ABB RAPID module: Projet1.mod

MODULE Lab1
! ----------------------------------------------------------------------------
! Programme : GPA546Lab1
! Auteurs : Olivier Millette ET Camilo Serna
! Date : Mai 14, 2024
! Révision : V0.0
!
! Description :
! Ce programme permet de prendre deux blocs dans une glissoire et de les
! superposer sur une table de travail.
! ----------------------------------------------------------------------------

  ! Donnees de type position enseignees
  PERS robtarget rGlissoire:=[[0,0,0],[1,0,0,0],[0,0,0,0],[9E+09,9E+09,9E+09,9E+09,9E+09,9E+09]];
  PERS robtarget rDepot:=[[0,0,0],[1,0,0,0],[0,0,0,0],[9E+09,9E+09,9E+09,9E+09,9E+09,9E+09]];
  PERS robtarget rRetrait:=[[0,0,0],[1,0,0,0],[0,0,0,0],[9E+09,9E+09,9E+09,9E+09,9E+09,9E+09]];

  ! Donnees de type position calculees
  VAR robtarget rDepot2;

  ! Donnees de type constante
  CONST num Epaisseur:= 1; ! Épaisseur d'un bloc (en pouces)
  CONST num PouceToMM:= 25.4; ! Facteur de conversion
  CONST num Decalage:= -80; ! Distance d'approche ou de retrait (mm) Additionnele(ajouter +X pour marge de sécurité)

  ! Données de type Variable
  VAR num EpaisMM:=0;

  ! Vitesse d'approche et de retrait (mm/sec)
  CONST speeddata LowSpeed:=[250,500,5000,1000];

  ! Vitesse maximale du robot (mm/sec)
  CONST speeddata HighSpeed:=[1000,500,5000,1000];

  ! Etat des entrees/sorties
  CONST dionum Ouverte:=0;
  CONST dionum Fermee:=1;
  CONST dionum Retracte:=0;
  CONST dionum Extension:=1;

  ! Variable pour limiter la zone de travail du robot
  VAR wztemporary EspaceRestreint;

! ----------------------------------------------------------------------------
! Procedure : main
! Auteurs : Yanick Noiseux
! Date : 4-08-2011
! Révision : 1.1
! Révision par: Martin Gaudreault
! Description :
! Routine qui est executee par le robot initialement.
! **** elle doit être en mode "cycle"
!
! ----------------------------------------------------------------------------
!**************************************************************************************
PROC main()

	! 1) Initialisation :
	init;

	! Deplacement a la position de repos
	MoveJ rRetrait, HighSpeed, fine, tPince_bloc\wobj:=wobj0;

	! 2) Calculs :
	EpaisMM := Epaisseur * PouceToMM; ! Conversion en mm
	rDepot2 := Offs(rDepot,0,0,-EpaisMM);

	! 3) Déplacement du premier bloc :
	! Prise du bloc dans le glissoire
	Prise;
	! Dépôt du bloc 1 à la localisation rDepot :
	Depot(rDepot);

	! 4) Déplacement du deuxième bloc :
	! Prise du bloc dans le glissoire
	Prise;
	! Dépôt du bloc 2 à la localisation rDepot :
	Depot(rDepot2);

	! 5) Retourner le robot a la position de repos
	MoveJ rRetrait, HighSpeed, fine, tPince_bloc\wobj:=wobj0;

	Pince\Ouvert; ! Ouvrir la pince

ENDPROC
!**************************************************************************************

! ----------------------------------------------------------------------------
! Procedure : init
! Auteurs : Yanick Noiseux
! Date : 4-08-2011
! Révision : 1.1
! Révision par: Martin Gaudreault
! Description :
! Routine qui initialise les variables systèmes et les états des sorties
!
! ----------------------------------------------------------------------------
!**************************************************************************************
PROC init()

	! volume pour limiter les articulation du robot
	VAR shapedata joint_space;

	! Ne garder que les deux constantes correspondant a votre robot
	! Ces valeurs ne doivent pas être changées afin d'aider a la securite et représentent
    ! les limites logicielles pour chacun des axes

	! *** décommentez ces deux lignes si vous êtes sur le robot 1
	!CONST jointtarget low_pos:=[[ 54, -25, -85, -90, -103, -289 ],[ 9E9, 9E9, 9E9, 9E9, 9E9, 9E9 ]];
	!CONST jointtarget high_pos:=[[ 128,  55,  55,  90,  103,  109 ],[ 9E9, 9E9, 9E9, 9E9, 9E9, 9E9 ]];

	! *** décommentez ces deux lignes si vous êtes sur le robot 2
	!CONST jointtarget low_pos:=[[ -134, -25, -85, -90, -103, -289 ],[ 9E9, 9E9, 9E9, 9E9, 9E9, 9E9 ]];
	!CONST jointtarget high_pos:=[[ -65,  55,  55,  90,  103,  109 ],[ 9E9, 9E9, 9E9, 9E9, 9E9, 9E9 ]];

	! *** décommentez ces deux lignes si vous êtes sur le robot 3
	!CONST jointtarget low_pos:=[[ 44, -25, -85, -90, -103, -289 ],[ 9E9, 9E9, 9E9, 9E9, 9E9, 9E9 ]];
	!CONST jointtarget high_pos:=[[ 118,  55,  55,  90,  103,  109 ],[ 9E9, 9E9, 9E9, 9E9, 9E9, 9E9 ]];

	! *** décommentez ces deux lignes si vous êtes sur le robot 4
	!CONST jointtarget low_pos:=[[ -104, -25, -85, -90, -103, -289 ],[ 9E9, 9E9, 9E9, 9E9, 9E9, 9E9 ]];
	!CONST jointtarget high_pos:=[[ -28,  55,  55,  90,  103,  109 ],[ 9E9, 9E9, 9E9, 9E9, 9E9, 9E9 ]];

	! activation de la limitation, obligatoire
	WZFree EspaceRestreint;
	WZLimJointDef \Outside, joint_space, low_pos, high_pos;
	WZLimSup \Temp, EspaceRestreint, joint_space;

	VelSet 25,1000; ! Limitation imposée pour la sécurité, obligatoire

	SetDO DO09_FV0101, Retracte; ! Rentrer le vérin
	Pince\Ouvert; ! Ouvrir la pince

ENDPROC
!**************************************************************************************

! ----------------------------------------------------------------------------
! Procedure : Prise
! Auteurs : Yanick Noiseux
! Date : 4-08-2011
! Révision : 1.0
!
! Description :
! Routine qui s'approche du glissoire, atends une piece,
! l'indexe et la prends de maniere securitaire
!
! ----------------------------------------------------------------------------
!**************************************************************************************
PROC Prise()

! Vérification de présence de bloc dans la glissoire
	IF DI09_ZS0101 = 0 THEN
		TPErase;
		TPWrite "Aucun bloc dans la glissoire";
		TPWrite "Placer deux bloc et remettre en mode AUTO";
		WaitDI DI09_ZS0101, 1; ! Attente d'un bloc
		Waittime 1; ! attente que le bloc se stabilise
	ENDIF

	! Prehension du bloc
	MoveJ RelTool(rGlissoire,0,0,Decalage),HighSpeed,z50,tPince_bloc\wobj:=wobj0;
	SetDO DO09_FV0101, Extension; ! Indexer le bloc durant le mouvement
	WAITDI DI14_ZS0104,1; ! Attendre pour le vérin sortie
	MoveL rGlissoire, LowSpeed, fine, tPince_bloc\wobj:=wobj0;
	Pince\Fermer; ! Fermer la pince
	SetDO DO09_FV0101, Retracte;
	WAITDI DI14_ZS0104,0;
	MoveL RelTool(rGlissoire,0,0,Decalage),LowSpeed,z50,tPince_bloc\wobj:=wobj0;

ENDPROC
!**************************************************************************************

! ----------------------------------------------------------------------------
! Procedure : Depot
! Auteurs : Yanick Noiseux
! Date : 4-08-2011
! Révision : 1.1
! Révision par: Martin Gaudreault
! Description :
! Routine qui initialise les variables systèmes et les états des sorties
!
! Parametre: recoit un robtarget où aller déposer le bloc avec aproche et degagement
!
! ----------------------------------------------------------------------------
!**************************************************************************************
PROC Depot(robtarget rPosDepot) 	! Déclaration de la procédure de dépôt
	! 1) Approche rapide à la position de dépôt, en décalant en Z pour éviter les collisions
	MoveJ RelTool(rPosDepot,0,0,Decalage), HighSpeed, z50, tPince_bloc\wobj:=wobj0;

	! 2) Descente linéaire en mode « fine » à vitesse réduite pour un positionnement précis
	MoveL rPosDepot, LowSpeed, fine, tPince_bloc;

	! 3) Ouverture de la pince pour relâcher le bloc
	Pince\Ouvert; ! Ouvrir la pince

	! 4) Remontée linéaire à la position d’approche (décalée en Z) pour dégager l’outil
	MoveL RelTool(rPosDepot,0,0,Decalage), LowSpeed, z50, tPince_bloc\wobj:=wobj0;

ENDPROC
!**************************************************************************************

! ----------------------------------------------------------------------------
! Procedure : Pince
! Auteurs : Yanick Noiseux
! Date : 4-08-2011
! Révision : 1.1
! Révision par: Martin Gaudreault
! Description :
! Routine qui Défini l'état de l'outil pince du robot
! ----------------------------------------------------------------------------
!**************************************************************************************
PROC Pince(\switch Ouvert | switch Fermer)

    ! Action sur la pince
    IF Present(Fermer) THEN
		! verifie si la sortie doit-être changé d'état
		IF Doutput(DO01_EE_PINCE01)=0 THEN
       		Set DO01_EE_PINCE01; ! Ferme la pince
			WAITTIME 1;  !  Attente que la pince bouge physiquement
		ENDIF
    ELSE
		! verifie si la sortie doit-être changé d'état
		IF Doutput(DO01_EE_PINCE01)=1 THEN
       		Reset DO01_EE_PINCE01; ! Ferme la pince
			WAITTIME 1;  !  Attente que la pince bouge physiquement
		ENDIF
    ENDIF

ENDPROC
!**************************************************************************************
ENDMODULE
